PROGRAM Descarga_semilla
VAR
	fbPE_B_VF1 :Equipo_Motor_ATV320;//Elevador embolse
	PE_B1_V1: Equipo_Valvula_5_2_biestable;
	PE_B1_V1_CmdAuto_Pos1:BOOL;
	PE_B1_V1_CmdAuto_Pos2:BOOL;
	PE_B2_V1: Equipo_Valvula_5_2_biestable;
	PE_B2_V1_CmdAuto_Pos1:BOOL;
	PE_B2_V1_CmdAuto_Pos2:BOOL;
	PE_B3_V1: Equipo_Valvula_5_2_biestable;
	PE_B3_V1_CmdAuto_Pos1:BOOL;
	PE_B3_V1_CmdAuto_Pos2:BOOL;
	PE_B1_V2_CmdAuto:BOOL;
	PE_B2_V2_CmdAuto:BOOL;
	PE_B3_V2_CmdAuto:BOOL;	
	
	bHS :BOOL;
	dintHS	:DINT:=3;
	Tmr_B1_LLS: TON;
	B1_LLS_Ok: BOOL;
	Tmr_B2_LLS: TON;
	B2_LLS_Ok: BOOL;
	TmrCicloCarga: TON;
	Cargar_B2: BOOL;
	AuxCargar_B2: BOOL;
	AuxB1_V1: BOOL;
	AuxB2_V1: BOOL;
	TmrDemoraB2_V1: TOF;
	TmrPE_B1_HLS: TON;	//Nível alto da caixa de sacarias
	TmrPE_B2_HLS: TON;	//Nível alto do BIGBAG 2
	TmrPE_B3_HLS: TON;	//Nível alto do BIGBAG 3
	TDemoraPE_B1_LLS: TON;
	TDemoraPE_BE2_LLS: TON;
	TDemoraPE_BE3_LLS: TON;
	Tmr_B3_LLS: TON;
	B3_LLS_Ok: BOOL;
	Tiempo_seg_to_TIME_PE_B_VF1: Tiempo_seg_to_TIME;
	TmrDemoraPE_B_VF1: TOF;
	TDemoraB3_V1: TOF;
	PE_B1_V1_Teste: Equipo_Valvula_5_2;
	PE_B1_V2_Teste: Equipo_Valvula_5_2;
	PE_B1_V3_Teste: Equipo_Valvula_5_2;
	TON_CaixaCheia: TON;
	PausaEnsaque: BOOL;	//Se as duas caixas de ensaque estiverem cheias e a descarga for no bigbag, pausa o processo
	// Atraso na descarga da caixa 3 para que não passem canecas cheias
	TOF_DescargaCX3: TOF;
END_VAR
VAR // added by the converter: edge detectors and wires of the graphical bodies
    _w1 : BOOL;
    _rt1 : R_TRIG;
END_VAR

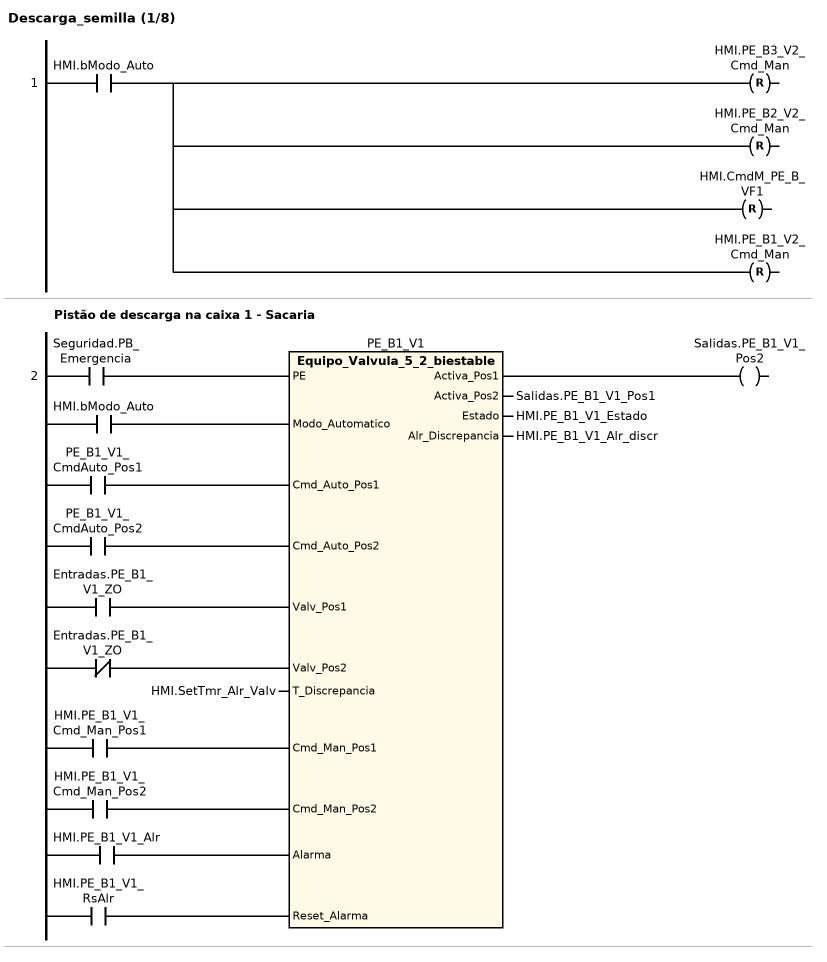
// NETWORK 1
_w1 := HMI.bModo_Auto;
HMI.PE_B3_V2_Cmd_Man R= _w1;
HMI.PE_B2_V2_Cmd_Man R= _w1;
HMI.CmdM_PE_B_VF1 R= _w1;
HMI.PE_B1_V2_Cmd_Man R= _w1;

// NETWORK 2: Pistão de descarga na caixa 1 - Sacaria
PE_B1_V1(
    PE := Seguridad.PB_Emergencia,
    Modo_Automatico := HMI.bModo_Auto,
    Cmd_Auto_Pos1 := PE_B1_V1_CmdAuto_Pos1,
    Cmd_Auto_Pos2 := PE_B1_V1_CmdAuto_Pos2,
    Valv_Pos1 := Entradas.PE_B1_V1_ZO,
    Valv_Pos2 := NOT Entradas.PE_B1_V1_ZO,
    T_Discrepancia := HMI.SetTmr_Alr_Valv,
    Cmd_Man_Pos1 := HMI.PE_B1_V1_Cmd_Man_Pos1,
    Cmd_Man_Pos2 := HMI.PE_B1_V1_Cmd_Man_Pos2,
    Alarma := HMI.PE_B1_V1_Alr,
    Reset_Alarma := HMI.PE_B1_V1_RsAlr,
    Activa_Pos2 => Salidas.PE_B1_V1_Pos1,
    Estado => HMI.PE_B1_V1_Estado,
    Alr_Discrepancia => HMI.PE_B1_V1_Alr_discr); // Equipo_Valvula_5_2_biestable
Salidas.PE_B1_V1_Pos2 := PE_B1_V1.Activa_Pos1;

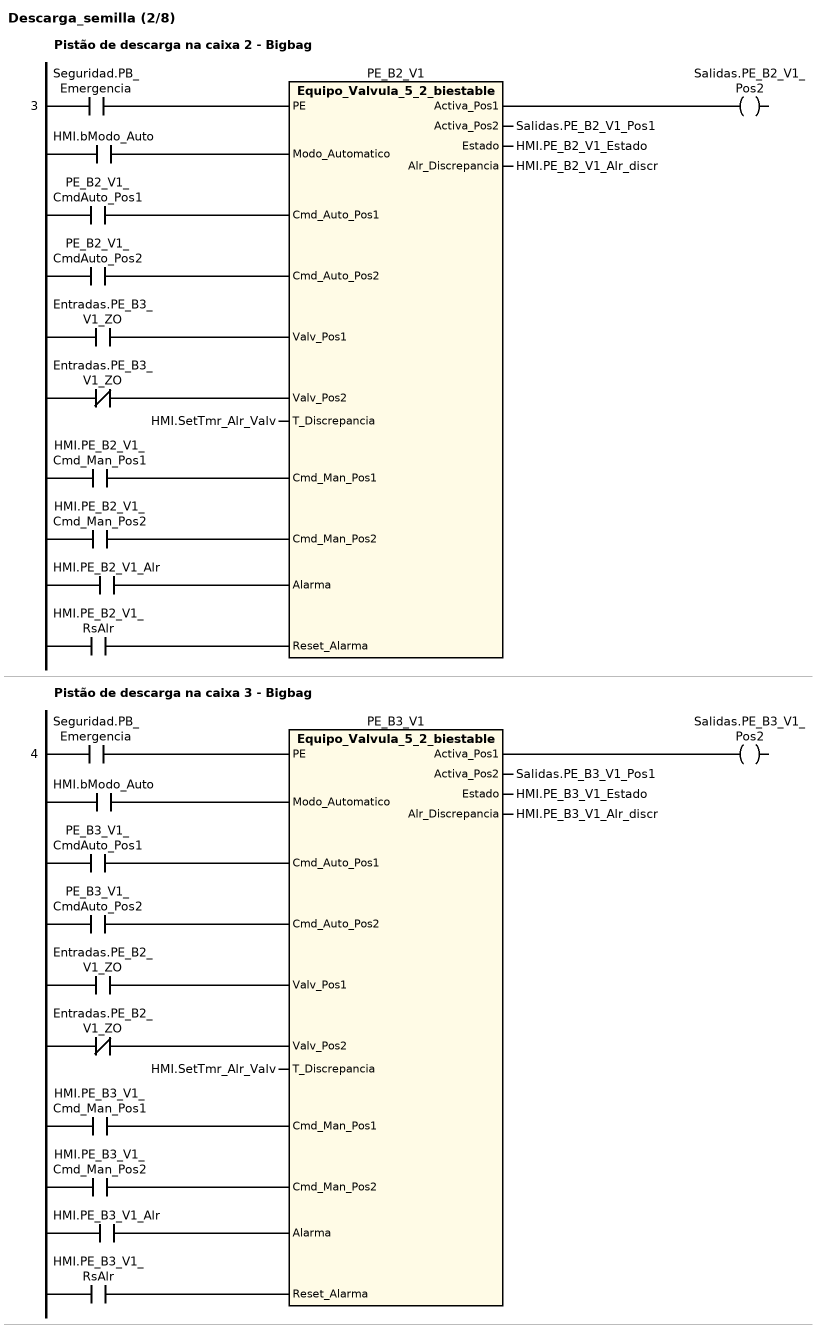
// NETWORK 3: Pistão de descarga na caixa 2 - Bigbag
PE_B2_V1(
    PE := Seguridad.PB_Emergencia,
    Modo_Automatico := HMI.bModo_Auto,
    Cmd_Auto_Pos1 := PE_B2_V1_CmdAuto_Pos1,
    Cmd_Auto_Pos2 := PE_B2_V1_CmdAuto_Pos2,
    Valv_Pos1 := Entradas.PE_B3_V1_ZO,
    Valv_Pos2 := NOT Entradas.PE_B3_V1_ZO,
    T_Discrepancia := HMI.SetTmr_Alr_Valv,
    Cmd_Man_Pos1 := HMI.PE_B2_V1_Cmd_Man_Pos1,
    Cmd_Man_Pos2 := HMI.PE_B2_V1_Cmd_Man_Pos2,
    Alarma := HMI.PE_B2_V1_Alr,
    Reset_Alarma := HMI.PE_B2_V1_RsAlr,
    Activa_Pos2 => Salidas.PE_B2_V1_Pos1,
    Estado => HMI.PE_B2_V1_Estado,
    Alr_Discrepancia => HMI.PE_B2_V1_Alr_discr); // Equipo_Valvula_5_2_biestable
Salidas.PE_B2_V1_Pos2 := PE_B2_V1.Activa_Pos1;

// NETWORK 4: Pistão de descarga na caixa 3 - Bigbag
PE_B3_V1(
    PE := Seguridad.PB_Emergencia,
    Modo_Automatico := HMI.bModo_Auto,
    Cmd_Auto_Pos1 := PE_B3_V1_CmdAuto_Pos1,
    Cmd_Auto_Pos2 := PE_B3_V1_CmdAuto_Pos2,
    Valv_Pos1 := Entradas.PE_B2_V1_ZO,
    Valv_Pos2 := NOT Entradas.PE_B2_V1_ZO,
    T_Discrepancia := HMI.SetTmr_Alr_Valv,
    Cmd_Man_Pos1 := HMI.PE_B3_V1_Cmd_Man_Pos1,
    Cmd_Man_Pos2 := HMI.PE_B3_V1_Cmd_Man_Pos2,
    Alarma := HMI.PE_B3_V1_Alr,
    Reset_Alarma := HMI.PE_B3_V1_RsAlr,
    Activa_Pos2 => Salidas.PE_B3_V1_Pos1,
    Estado => HMI.PE_B3_V1_Estado,
    Alr_Discrepancia => HMI.PE_B3_V1_Alr_discr); // Equipo_Valvula_5_2_biestable
Salidas.PE_B3_V1_Pos2 := PE_B3_V1.Activa_Pos1;

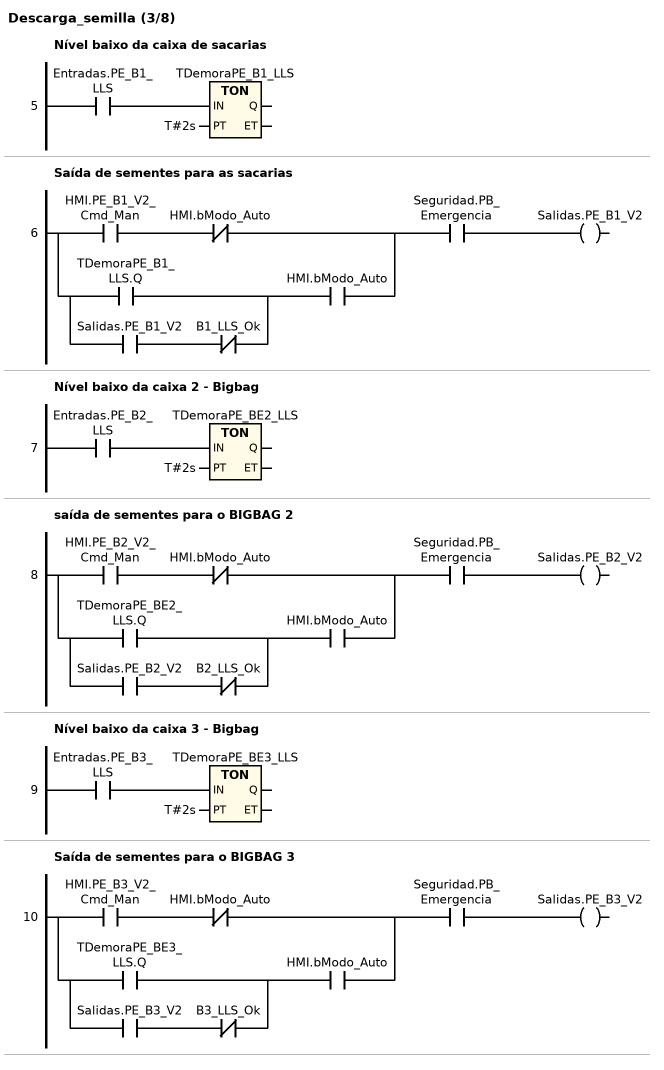
// NETWORK 5: Nível baixo da caixa de sacarias
TDemoraPE_B1_LLS(IN := Entradas.PE_B1_LLS, PT := T#2s); // TON

// NETWORK 6: Saída de sementes para as sacarias
Salidas.PE_B1_V2 := (HMI.PE_B1_V2_Cmd_Man AND NOT HMI.bModo_Auto OR (TDemoraPE_B1_LLS.Q OR Salidas.PE_B1_V2 AND NOT B1_LLS_Ok) AND HMI.bModo_Auto) AND Seguridad.PB_Emergencia;

// NETWORK 7: Nível baixo da caixa 2 - Bigbag
TDemoraPE_BE2_LLS(IN := Entradas.PE_B2_LLS, PT := T#2s); // TON

// NETWORK 8: saída de sementes para o BIGBAG 2
Salidas.PE_B2_V2 := (HMI.PE_B2_V2_Cmd_Man AND NOT HMI.bModo_Auto OR (TDemoraPE_BE2_LLS.Q OR Salidas.PE_B2_V2 AND NOT B2_LLS_Ok) AND HMI.bModo_Auto) AND Seguridad.PB_Emergencia;

// NETWORK 9: Nível baixo da caixa 3 - Bigbag
TDemoraPE_BE3_LLS(IN := Entradas.PE_B3_LLS, PT := T#2s); // TON

// NETWORK 10: Saída de sementes para o BIGBAG 3
Salidas.PE_B3_V2 := (HMI.PE_B3_V2_Cmd_Man AND NOT HMI.bModo_Auto OR (TDemoraPE_BE3_LLS.Q OR Salidas.PE_B3_V2 AND NOT B3_LLS_Ok) AND HMI.bModo_Auto) AND Seguridad.PB_Emergencia;

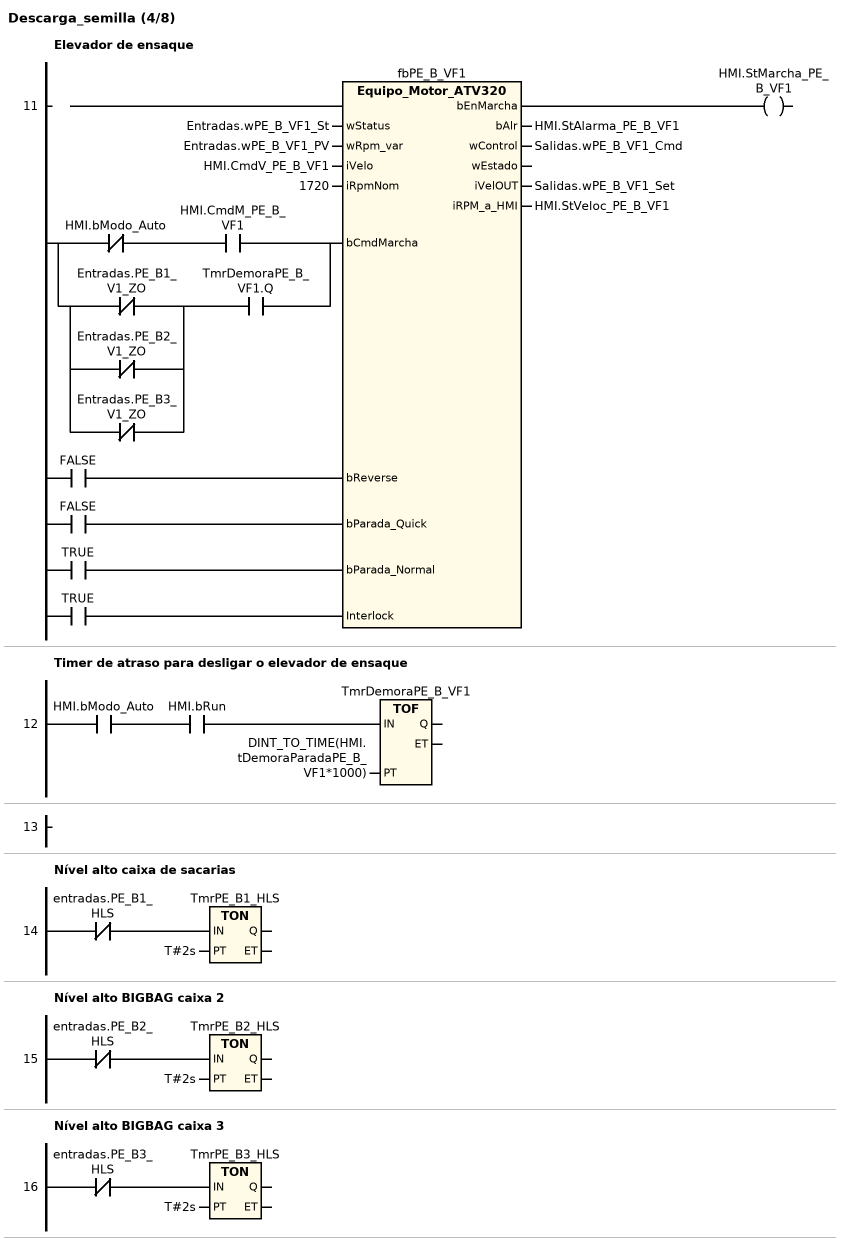
// NETWORK 11: Elevador de ensaque
fbPE_B_VF1(
    wStatus := Entradas.wPE_B_VF1_St,
    wRpm_var := Entradas.wPE_B_VF1_PV,
    iVelo := HMI.CmdV_PE_B_VF1,
    iRpmNom := 1720,
    bCmdMarcha := NOT HMI.bModo_Auto AND HMI.CmdM_PE_B_VF1 OR (NOT Entradas.PE_B1_V1_ZO OR NOT Entradas.PE_B2_V1_ZO OR NOT Entradas.PE_B3_V1_ZO) AND TmrDemoraPE_B_VF1.Q,
    bReverse := FALSE,
    bParada_Quick := FALSE,
    bParada_Normal := TRUE,
    Interlock := TRUE,
    bAlr => HMI.StAlarma_PE_B_VF1,
    wControl => Salidas.wPE_B_VF1_Cmd,
    iVelOUT => Salidas.wPE_B_VF1_Set,
    iRPM_a_HMI => HMI.StVeloc_PE_B_VF1); // Equipo_Motor_ATV320
HMI.StMarcha_PE_B_VF1 := fbPE_B_VF1.bEnMarcha;

// NETWORK 12: Timer de atraso para desligar o elevador de ensaque
TmrDemoraPE_B_VF1(IN := HMI.bModo_Auto AND HMI.bRun, PT := DINT_TO_TIME(HMI.tDemoraParadaPE_B_VF1*1000)); // TOF

// NETWORK 13

// NETWORK 14: Nível alto caixa de sacarias
TmrPE_B1_HLS(IN := NOT entradas.PE_B1_HLS, PT := T#2s); // TON

// NETWORK 15: Nível alto BIGBAG caixa 2
TmrPE_B2_HLS(IN := NOT entradas.PE_B2_HLS, PT := T#2s); // TON

// NETWORK 16: Nível alto BIGBAG caixa 3
TmrPE_B3_HLS(IN := NOT entradas.PE_B3_HLS, PT := T#2s); // TON

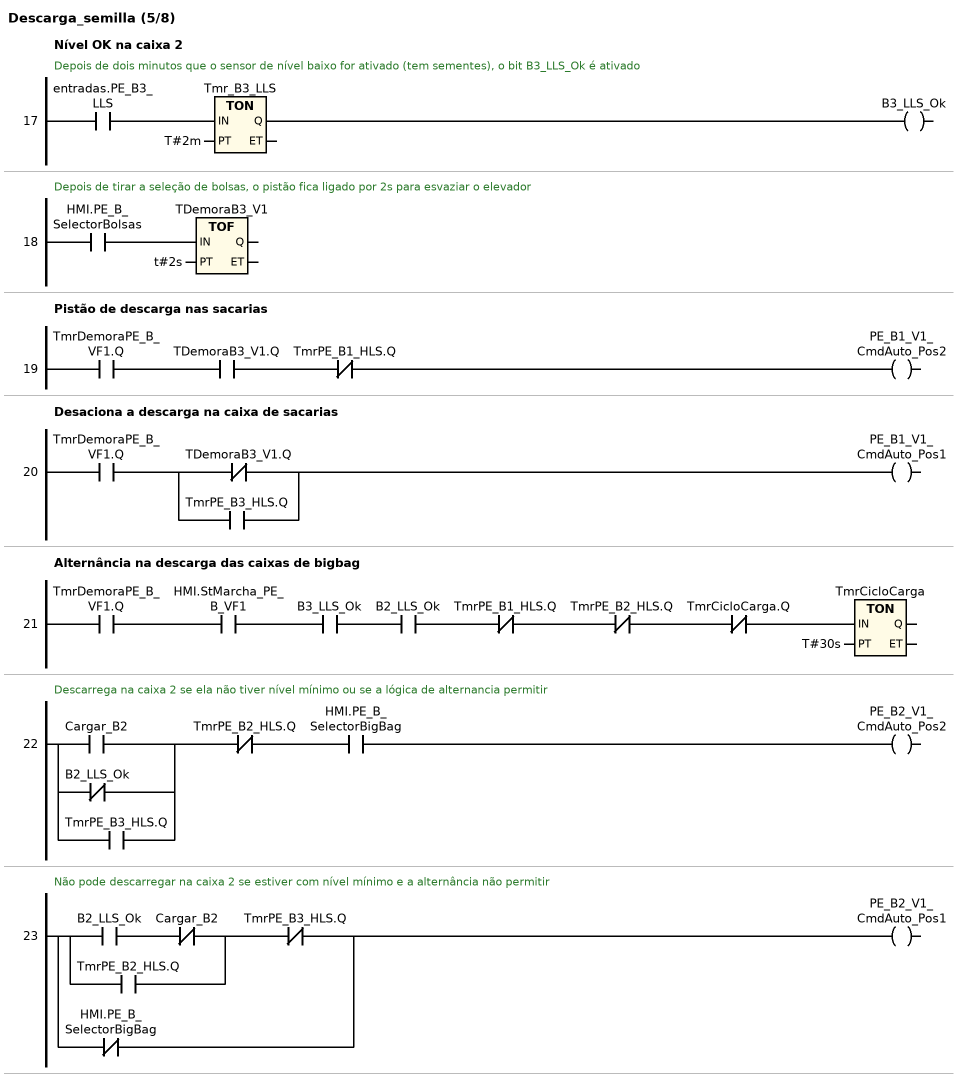
// NETWORK 17: Nível OK na caixa 2
// Depois de dois minutos que o sensor de nível baixo for ativado (tem sementes), o bit B3_LLS_Ok é ativado
Tmr_B3_LLS(IN := entradas.PE_B3_LLS, PT := T#2m); // TON
B3_LLS_Ok := Tmr_B3_LLS.Q;

// NETWORK 18
// Depois de tirar a seleção de bolsas, o pistão fica ligado por 2s para esvaziar o elevador
TDemoraB3_V1(IN := HMI.PE_B_SelectorBolsas, PT := t#2s); // TOF

// NETWORK 19: Pistão de descarga nas sacarias
PE_B1_V1_CmdAuto_Pos2 := TmrDemoraPE_B_VF1.Q AND TDemoraB3_V1.Q AND NOT TmrPE_B1_HLS.Q;

// NETWORK 20: Desaciona a descarga na caixa de sacarias
PE_B1_V1_CmdAuto_Pos1 := TmrDemoraPE_B_VF1.Q AND (NOT TDemoraB3_V1.Q OR TmrPE_B3_HLS.Q);

// NETWORK 21: Alternância na descarga das caixas de bigbag
TmrCicloCarga(IN := TmrDemoraPE_B_VF1.Q AND HMI.StMarcha_PE_B_VF1 AND B3_LLS_Ok AND B2_LLS_Ok AND NOT TmrPE_B1_HLS.Q AND NOT TmrPE_B2_HLS.Q AND NOT TmrCicloCarga.Q, PT := T#30s); // TON

// NETWORK 22
// Descarrega na caixa 2 se ela não tiver nível mínimo ou se a lógica de alternancia permitir
PE_B2_V1_CmdAuto_Pos2 := (Cargar_B2 OR NOT B2_LLS_Ok OR TmrPE_B3_HLS.Q) AND NOT TmrPE_B2_HLS.Q AND HMI.PE_B_SelectorBigBag;

// NETWORK 23
// Não pode descarregar na caixa 2 se estiver com nível mínimo e a alternância não permitir
PE_B2_V1_CmdAuto_Pos1 := (B2_LLS_Ok AND NOT Cargar_B2 OR TmrPE_B2_HLS.Q) AND NOT TmrPE_B3_HLS.Q OR NOT HMI.PE_B_SelectorBigBag;

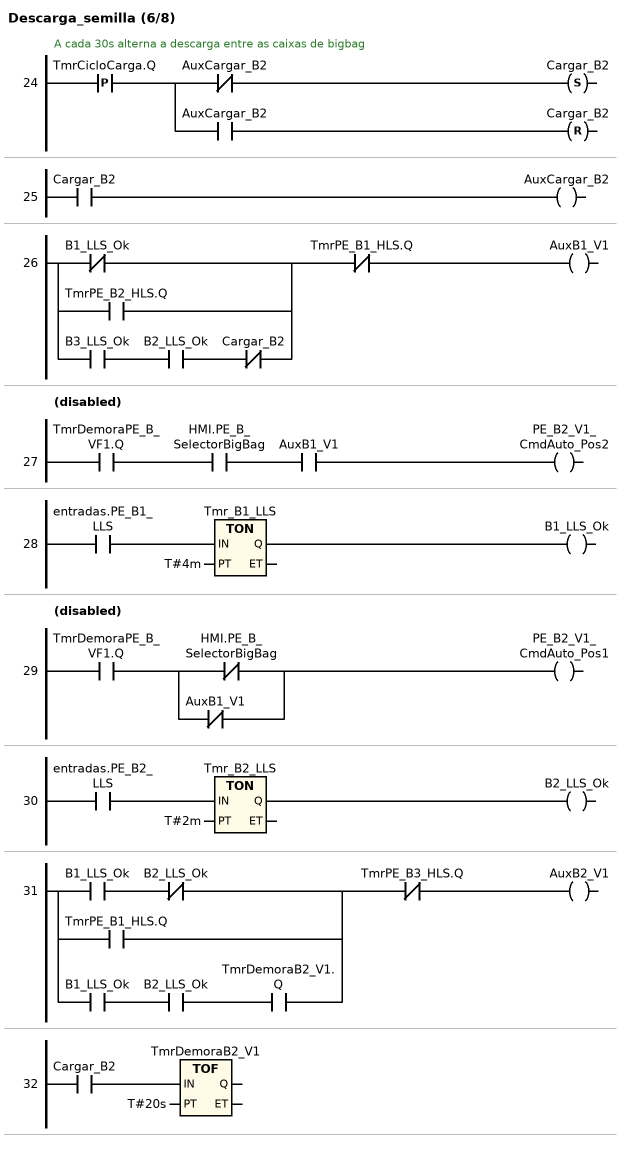
// NETWORK 24
// A cada 30s alterna a descarga entre as caixas de bigbag
_rt1(CLK := TmrCicloCarga.Q);
Cargar_B2 S= _rt1.Q AND NOT AuxCargar_B2;
Cargar_B2 R= _rt1.Q AND AuxCargar_B2;

// NETWORK 25
AuxCargar_B2 := Cargar_B2;

// NETWORK 26
AuxB1_V1 := (NOT B1_LLS_Ok OR TmrPE_B2_HLS.Q OR B3_LLS_Ok AND B2_LLS_Ok AND NOT Cargar_B2) AND NOT TmrPE_B1_HLS.Q;

// NETWORK 27 (disabled)
// PE_B2_V1_CmdAuto_Pos2 := TmrDemoraPE_B_VF1.Q AND HMI.PE_B_SelectorBigBag AND AuxB1_V1;

// NETWORK 28
Tmr_B1_LLS(IN := entradas.PE_B1_LLS, PT := T#4m); // TON
B1_LLS_Ok := Tmr_B1_LLS.Q;

// NETWORK 29 (disabled)
// PE_B2_V1_CmdAuto_Pos1 := TmrDemoraPE_B_VF1.Q AND (NOT HMI.PE_B_SelectorBigBag OR NOT AuxB1_V1);

// NETWORK 30
Tmr_B2_LLS(IN := entradas.PE_B2_LLS, PT := T#2m); // TON
B2_LLS_Ok := Tmr_B2_LLS.Q;

// NETWORK 31
AuxB2_V1 := (B1_LLS_Ok AND NOT B2_LLS_Ok OR TmrPE_B1_HLS.Q OR B1_LLS_Ok AND B2_LLS_Ok AND TmrDemoraB2_V1.Q) AND NOT TmrPE_B3_HLS.Q;

// NETWORK 32
TmrDemoraB2_V1(IN := Cargar_B2, PT := T#20s); // TOF

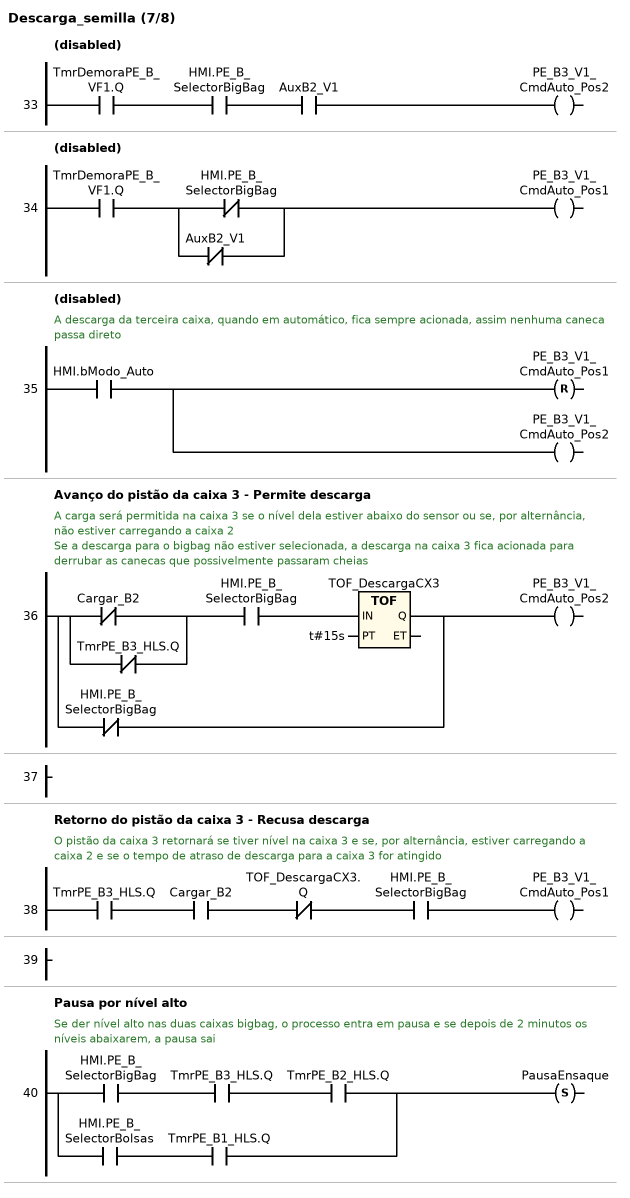
// NETWORK 33 (disabled)
// PE_B3_V1_CmdAuto_Pos2 := TmrDemoraPE_B_VF1.Q AND HMI.PE_B_SelectorBigBag AND AuxB2_V1;

// NETWORK 34 (disabled)
// PE_B3_V1_CmdAuto_Pos1 := TmrDemoraPE_B_VF1.Q AND (NOT HMI.PE_B_SelectorBigBag OR NOT AuxB2_V1);

// NETWORK 35 (disabled)
// A descarga da terceira caixa, quando em automático, fica sempre acionada, assim nenhuma caneca passa direto
// PE_B3_V1_CmdAuto_Pos1 R= HMI.bModo_Auto;
// PE_B3_V1_CmdAuto_Pos2 := HMI.bModo_Auto;

// NETWORK 36: Avanço do pistão da caixa 3 - Permite descarga
// A carga será permitida na caixa 3 se o nível dela estiver abaixo do sensor ou se, por alternância, não estiver carregando a caixa 2
// Se a descarga para o bigbag não estiver selecionada, a descarga na caixa 3 fica acionada para derrubar as canecas que possivelmente passaram cheias
TOF_DescargaCX3(IN := (NOT Cargar_B2 OR NOT TmrPE_B3_HLS.Q) AND HMI.PE_B_SelectorBigBag, PT := t#15s); // TOF
PE_B3_V1_CmdAuto_Pos2 := TOF_DescargaCX3.Q OR NOT HMI.PE_B_SelectorBigBag;

// NETWORK 37

// NETWORK 38: Retorno do pistão da caixa 3 - Recusa descarga
// O pistão da caixa 3 retornará se tiver nível na caixa 3 e se, por alternância, estiver carregando a caixa 2 e se o tempo de atraso de descarga para a caixa 3 for atingido
PE_B3_V1_CmdAuto_Pos1 := TmrPE_B3_HLS.Q AND Cargar_B2 AND NOT TOF_DescargaCX3.Q AND HMI.PE_B_SelectorBigBag;

// NETWORK 39

// NETWORK 40: Pausa por nível alto
// Se der nível alto nas duas caixas bigbag, o processo entra em pausa e se depois de 2 minutos os níveis abaixarem, a pausa sai
PausaEnsaque S= HMI.PE_B_SelectorBigBag AND TmrPE_B3_HLS.Q AND TmrPE_B2_HLS.Q OR HMI.PE_B_SelectorBolsas AND TmrPE_B1_HLS.Q;

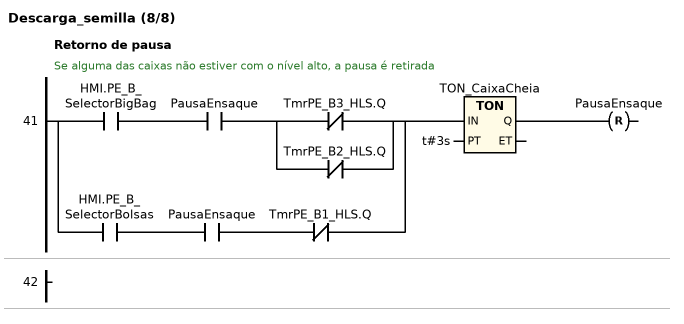
// NETWORK 41: Retorno de pausa
// Se alguma das caixas não estiver com o nível alto, a pausa é retirada
TON_CaixaCheia(IN := HMI.PE_B_SelectorBigBag AND PausaEnsaque AND (NOT TmrPE_B3_HLS.Q OR NOT TmrPE_B2_HLS.Q) OR HMI.PE_B_SelectorBolsas AND PausaEnsaque AND NOT TmrPE_B1_HLS.Q, PT := t#3s); // TON
PausaEnsaque R= TON_CaixaCheia.Q;

// NETWORK 42

END_PROGRAM

(* stored: Version 1.1.0.1, ProductVersion 3.1.4024.14
   POU Descarga_semilla: Id {9a4fee84-3989-467f-9645-5f5319af8c88}, SpecialFunc None *)
